TYPE IdHandle_t : POINTER TO ObjectId_t; END_TYPE

(* stored: Version 1.1.0.1, ProductVersion 3.1.4024.12
   DUT IdHandle_t: Id {c682234d-c852-4043-b036-188aefbbf4b8} *)
